FUNCTION AdditionFunction : REAL
VAR_INPUT
	i_valueA : REAL;
	i_valueB : REAL;
END_VAR

AdditionFunction := i_valueA + i_valueB;

END_FUNCTION

(* stored: Version 1.1.0.1, ProductVersion 3.1.4022.12
   POU AdditionFunction: Id {038f9d96-1cd4-4a69-88de-008e482696ef}, SpecialFunc None *)
